// TIA Portal V19 export
TYPE "TO_Diagnostic"
// stored: Access Published
   STRUCT
      DeviceType : Int;   // Device type for HMI diagnostic (see manual)
      ErrorReached_SwLimitMinus : Bool;
      ErrorReached_SwLimitPlus : Bool;
      ErrorReached_HwLimitMinus : Bool;
      ErrorReached_HwLimitPlus : Bool;
      ErrorMC_Reset : Bool;
      ErrorMC_Power : Bool;
      ErrorMC_Home : Bool;
      ErrorMC_MoveVel : Bool;
      ErrorMC_MoveAbs : Bool;
      ErrorMC_GearIn : Bool;
      ErrorMC_GearInPos : Bool;
      ErrorMC_CamIn : Bool;
      ErrorMC_Halt : Bool;
      ErrorMC_Stop : Bool;
      ErrorMC_AbortMeas : Bool;
      ErrorMC_MeasInp : Bool;
      ErrorMC_MoveSuperImp : Bool;
      ErrorMC_MoveLinearAbs : Bool;
      ErrorMC_SetWorkSpaceZoneActive : Bool;
      ErrorMC_SetWorkSpaceZoneInactive : Bool;
      ErrorMC_SetKinematicsZoneActive : Bool;
      ErrorMC_SetKinematicsZoneInactive : Bool;
      ErrorMC_GroupStop : Bool;
      ErrorMC_SetTool : Bool;
      MC_ErrorPresence : Bool;   // MC Error presence
      MC_Message : Word;   // Message form an MC Function
      TO_SimulationActive : Bool;   // Technology object simulation active
      TO_RestartNeeded : Bool;   // Restart technology object needed
      TO_RestartActive : Bool;   // Restart technology object active
      TO_RestartEnable : Bool;   // Restart technology object enabled
      TO_RestartCmd : Bool;   // Restart technology object command
      TO_ErrorPresence : Bool;   // Technology object error presence
      TO_Message : UDInt;   // Message from technology object
      Drive_ErrorPresence : Bool;   // Drive error presence
      Drive_Message : UInt;   // Message from Drive
      MessageType : Int;   // 0=NoMessage, 1=Warning, 2=Alarm
   END_STRUCT;
END_TYPE
